{attribute 'enable_dynamic_creation'}
FUNCTION_BLOCK FutureMCMoveAbsolute EXTENDS FB_AbstructFuture
VAR_INPUT
END_VAR
VAR_OUTPUT
END_VAR
VAR
	_fb_move_abs	: MC_MoveAbsolute;
	_executor		: FB_Executor;
	_axis: REFERENCE TO AXIS_REF;
	_position : MC_LREAL;
	_velocity : MC_LREAL;
	_acceleration: MC_LREAL;
	_deceleration: MC_LREAL;
	_jerk		: MC_LREAL;
	_option : ST_MoveOptions;
	_buffer_mode : MC_BufferMode ;
	_error_id :UDINT;
	_exec_state : UDINT;
	_abort_state : UINT;
END_VAR

METHOD abort : BOOL // Return TRUE if finish.
VAR_INST
	future_halt : FutureMcHalt;
END_VAR
CASE _abort_state OF
	0:
		_exec_state := 0;
		future_halt.set_parameters(_axis, _deceleration, _jerk);
		future_halt.future_name := 'HALT MOVE_RELATIVE';
		_executor.future := future_halt;
		_abort_state := 1;
	1:
		IF _executor.execute() AND _executor.nErrorID = 0 THEN
			_abort_state := 2;
		END_IF
		
		IF _executor.current_state = E_FutureExecutionState.wait_for_process THEN
			_executor.start();
		END_IF
	2:
		abort := TRUE;
END_CASE
END_METHOD

METHOD execute : BOOL // Return TRUE if finish.

CASE _exec_state OF
	0:
		_abort_state := 0;
		_fb_move_abs(Axis := _axis,Execute := FALSE);
		_fb_move_abs(
			Execute := TRUE,
			Axis := _axis,
			Position := _position,
			Velocity := _velocity,
			Acceleration := _acceleration,
			Deceleration := _deceleration,
			Jerk := _jerk,
			BufferMode := _buffer_mode,
			Options := _option
		);
		_exec_state := 1;
	1:
		IF _fb_move_abs.Busy THEN
			_fb_move_abs(Axis := _axis,Execute := FALSE);
		END_IF
END_CASE

_error_id := _fb_move_abs.ErrorID;
execute := _fb_move_abs.Done OR _fb_move_abs.Error;
END_METHOD

METHOD init : BOOL // Return TRUE if finish.

VAR
	axis: INT;
END_VAR
_exec_state := 0;
_abort_state := 0;
_error_id := _fb_move_abs.ErrorID;
init := TRUE;
END_METHOD

PROPERTY nErrorID : UDINT
GET
nErrorID := _error_id;
END_GET
SET
END_SET
END_PROPERTY

METHOD set_options : BOOL
VAR_INPUT
	option : ST_MoveOptions;
END_VAR
_option := option;
END_METHOD

METHOD set_parameters : BOOL
VAR_INPUT
	axis : REFERENCE TO AXIS_REF;
	position : MC_LREAL;
	velocity : MC_LREAL;
	acceleration	: MC_LREAL;		// Set deceleration in case let moving axis halt.
	deceleration	: MC_LREAL;		// Set deceleration in case let moving axis halt.
	jerk			: MC_LREAL;		// Set jerk in case let moving axis halt.
	buffer_mode : MC_BufferMode;
END_VAR
_axis REF= axis;
_position := position;
_velocity := velocity;
_acceleration := acceleration;
_deceleration := deceleration;
_jerk := jerk;
_buffer_mode := buffer_mode;
END_METHOD

END_FUNCTION_BLOCK

(* stored: Version 1.1.0.1, ProductVersion 3.1.4024.12
   POU FutureMCMoveAbsolute: Id {79bb57a1-f47d-4bcf-938a-520a06e0174a}, SpecialFunc None
   Method abort: Id {d55adceb-96cc-4338-86fc-114b02148736}
   Method execute: Id {04bb725d-9f81-4860-b243-c8cff20c19f8}
   Method init: Id {69b400a8-eed4-45f3-ae8d-2adfc6cc9d75}
   Property nErrorID: Id {dcbea886-840a-4451-a8f6-dbc15161fed0}
   Get Get: Id {ec03a1e5-2940-42ad-8905-125646af9c0f}
   Set Set: Id {5583237f-05f5-42b5-a279-dc47e285a901}
   Method set_options: Id {f1d5c719-e65a-4eae-bbe5-a4bda3562ddf}
   Method set_parameters: Id {d0fa521f-94a0-4187-b05e-77f37bff19ee} *)
